// TwinCAT 3 PLC project Untitled1
// ProgramVersion: 3.1.4024.0
// libraries:
//   Tc2_Standard, * (Beckhoff Automation GmbH)
//   Tc2_System, * (Beckhoff Automation GmbH)
//   Tc3_Module, * (Beckhoff Automation GmbH)
// project tree:
//   GVLs/ GVL.TcGVL
//   / PlcTask.TcTTO
//   POUs/ FB_M.TcPOU, FB_S.TcPOU, MAIN.TcPOU

CONFIGURATION Untitled1
    RESOURCE PLC ON TwinCAT3
        TASK PlcTask(INTERVAL := T#10ms, PRIORITY := 20);
        PROGRAM MAIN WITH PlcTask : MAIN;
    END_RESOURCE
END_CONFIGURATION

// ---- GVLs/GVL.TcGVL
{attribute 'qualified_only'}
VAR_GLOBAL CONSTANT
	tValveOffTimer		:TIME := T#10S;
	tValveOnTimer		:TIME := T#5S;
	
END_VAR
VAR_GLOBAL
	//Sensors
	bLowSensor			:BOOL := TRUE;	//LV, 
	bHighSensor			:BOOL;			//HV
	bHeatRelay			:BOOL; 			//TH
	bTankEmpty			:BOOL;			//UT
	
	//Manual Input Switch
	bManualMotor				:BOOL;
	bManualValve				:BOOL;

END_VAR

// ---- POUs/MAIN.TcPOU
PROGRAM MAIN
VAR
	fbMotor			:FB_M;
	fbValve			:FB_S;
END_VAR

fbMotor();
fbValve	();

END_PROGRAM

// ---- POUs/FB_M.TcPOU
FUNCTION_BLOCK FB_M
VAR_INPUT	
END_VAR
VAR_OUTPUT
	bMotor				:BOOL;			//KM
END_VAR
VAR
	bMotorOnButton		:BOOL;			//MB
	bMotorOffButton		:BOOL;			//MK
	bPrevOn				:BOOL;
	bPrevOff			:BOOL;

	nState				:UDINT:=0;		//0:Default, 20:Autorun, 40:Manual
END_VAR

CASE nState OF
	0:	//Stand by
		IF NOT GVL.bHeatRelay AND NOT GVL.bHighSensor THEN
			IF	GVL.bLowSensor THEN
				nState := 20;
			ELSIF GVL.bManualMotor THEN
				nState := 40;
			ELSE
				nState := 0;
				bMotor := 0;
			END_IF
		ELSE
			bMotor := FALSE;
			nState := 0;	
		END_IF
			
	20:
		bMotor := TRUE;
		
		IF GVL.bManualMotor THEN
			nState := 40;
		ELSE
			nState := 0;
		END_IF
	
	40:
		IF (bMotorOnButton AND NOT bPrevOn) THEN
			bMotorOffButton:=FALSE;
			bMotor := TRUE;
		ELSIF (bMotorOffButton AND NOT bPrevOff) THEN
			bMotorOnButton:=FALSE;
			bMotor := FALSE;		
		END_IF
		
		bPrevOn := bMotorOnButton;
		bPrevOff := bMotorOffButton;
		
		IF NOT GVL.bManualMotor THEN
			nState := 0;
		ELSE
			nState := 40;
		END_IF
		
		//state visszavezetés
	
END_CASE

END_FUNCTION_BLOCK

// ---- POUs/FB_S.TcPOU
FUNCTION_BLOCK FB_S
VAR_INPUT

END_VAR
VAR_OUTPUT
	bValve				:BOOL;
END_VAR
VAR
	bValveOpen			:BOOL;	//SB Testing TRUE
	bValveClosed		:BOOL;	//SK
	bPrevOpen			:BOOL;
	bPrevClosed			:BOOL;	

	//on/off buttons or every 90 sec for 30sec if tank not empty
	nState				:UDINT := 0; //0: Default, 20: Autorun 40: Manual
	myTimer				:TON;
	tCurrentTime		:TIME;
	bTemp				:BOOL;
END_VAR

CASE nState OF
	0: //Scanning for Errors
		IF GVL.bHeatRelay OR GVL.bTankEmpty THEN
			//Error log
			bValve := FALSE;
			nState := 0;		//Stay in standby state 0
		ELSE
			nState := 20;
		END_IF
	20:	//Auto Closed
		IF GVL.bManualValve THEN
			nState := 60;
		END_IF;
		tCurrentTime := GVL.tValveOffTimer;
		bValve := FALSE;
		IF myTimer.Q THEN
			nState := 40;	
			myTimer(IN := FALSE);
		END_IF
	40: //Auto Open
		IF GVL.bManualValve THEN
			nState := 60;
		END_IF;
		tCurrentTime := GVL.tValveOnTimer;
		bValve := TRUE;
		IF myTimer.Q THEN
			nState := 0;
			myTimer(IN := FALSE);
		END_IF
		
	60:
		IF (bValveOpen AND NOT bPrevOpen) THEN
			bValveClosed:=FALSE;
			bValve := TRUE;
		ELSIF (BValveClosed AND NOT bPrevClosed) THEN
			BValveOpen:=FALSE;
			bValve := FALSE;		
		END_IF
		
		bPrevOpen := bValveOpen;
		bPrevClosed := bValveClosed;		
		
		IF NOT GVL.bManualValve THEN
			nState := 0;
		ELSE
			nState := 60;
		END_IF
END_CASE

myTimer(IN:=TRUE, PT:=tCurrentTime);
myTimer(IN:=TRUE, PT:=tCurrentTime);

END_FUNCTION_BLOCK
